(* CoDeSys 2.3 export: MODBUS_FBD.EXP *)

(* POU modbus_FBD, FBD *)
PROGRAM modbus_FBD
VAR
	get1_modbus: MB_RD_HOLD_REGS;    (*функция 03 - чтение параметра типа INT*)
	get2_modbus: MB_RD_INP_REGS;		(*функция 04 - чтение трех параметров типа INT*)
	get3_modbus: MB_RD_HOLD_REGS;	(*функция 03 - чтение параметра типа Float*)
	COM_SERVICE1: COM_SERVICE;		(*функция открытия COM-порта*)

	Buffer: ARRAY[0..255] OF BYTE;		(* байтовый буфер данных *)
     	cmpl: BOOL;
	port_opened:  BYTE := 0;
	Init: BOOL;								(* признак инициализации пользовательской программы *)
	Settings:COMSETTINGS;				(* настройки последовательного порта *)
      	com_num: PORTS:=0;				(*0 - RS-485, 1 - RS-232*)
	enabl: BOOL;							(*состояние работы блока*)
	err: INT;								(*номер ошибки*)
	TimeOut: TIME:=T#50ms;				(*таймаут*)
	Exception: BYTE;
	DataSize: WORD;
	master1: BYTE:= 0;

	x:WORD;						(*считанное значение*)
	x1: WORD;						(*переменная для записи по сети*)
	x2: WORD;						(*переменная для записи по сети*)
	x3: WORD;						(*переменная для записи по сети*)
	d:  REAL;						(*считанное значение*)
	ptr_D:POINTER TO BYTE;

	ctu1: CTU;
	a: BOOL;
	ynjj: BOOL;
END_VAR
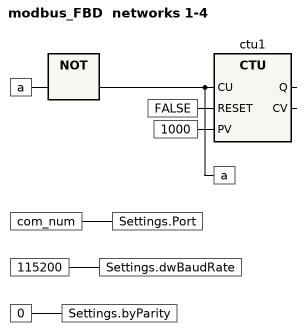
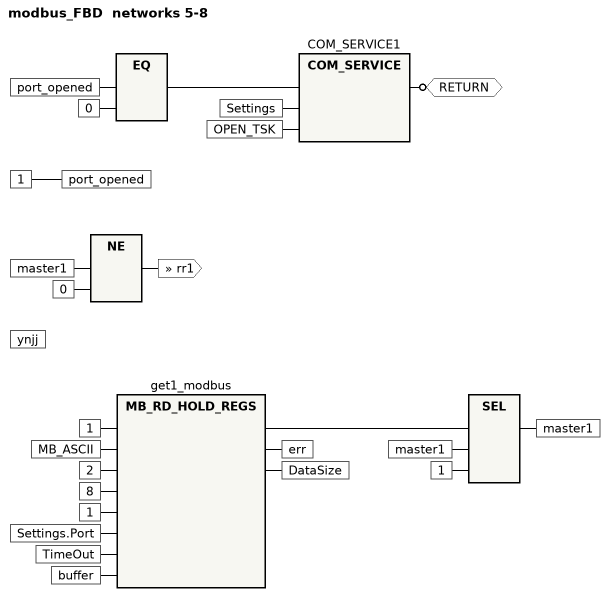
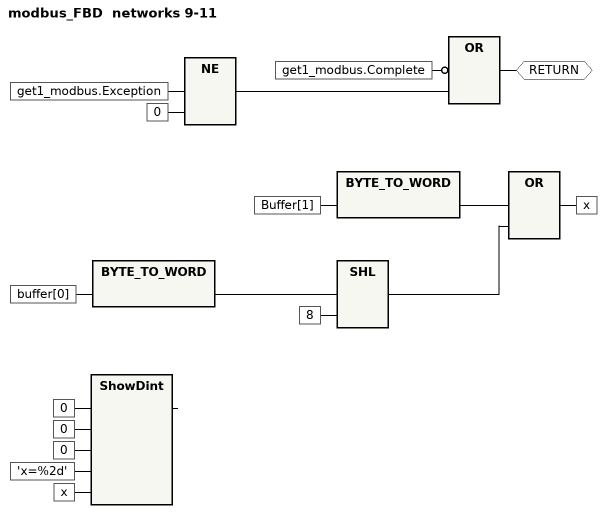
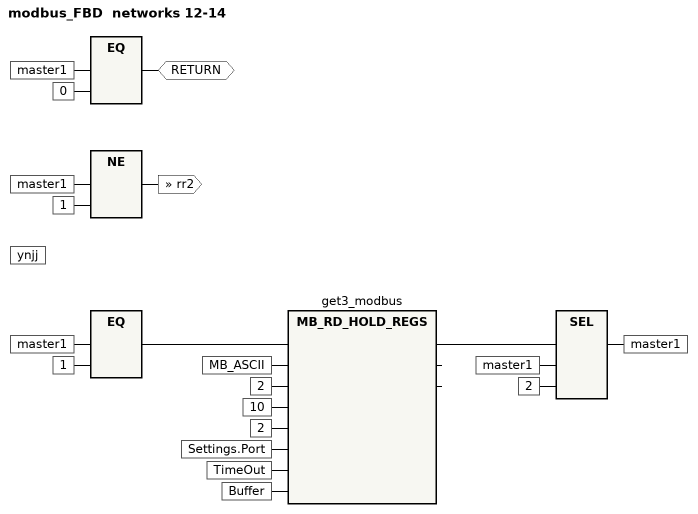
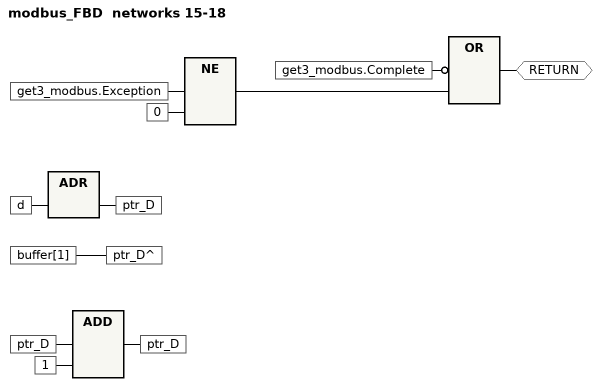
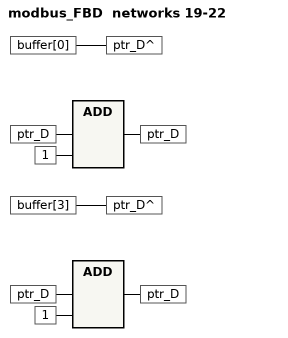
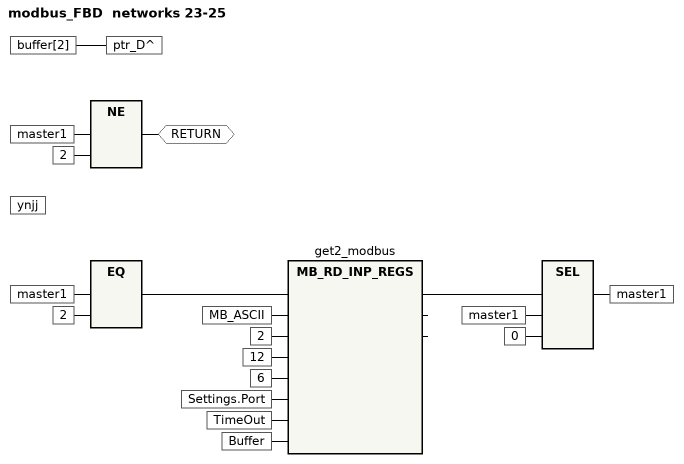
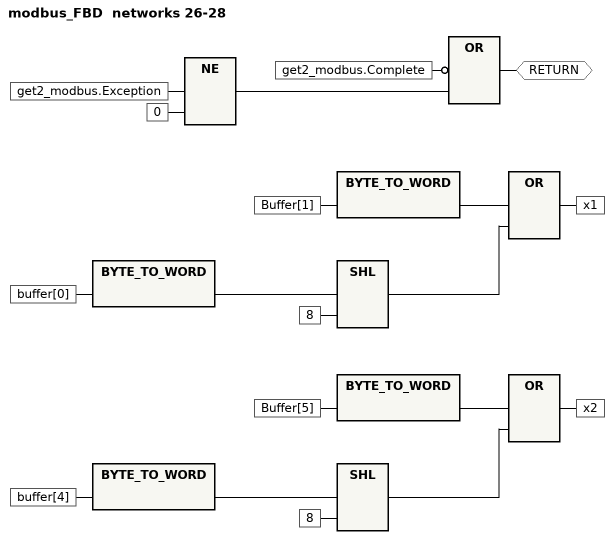
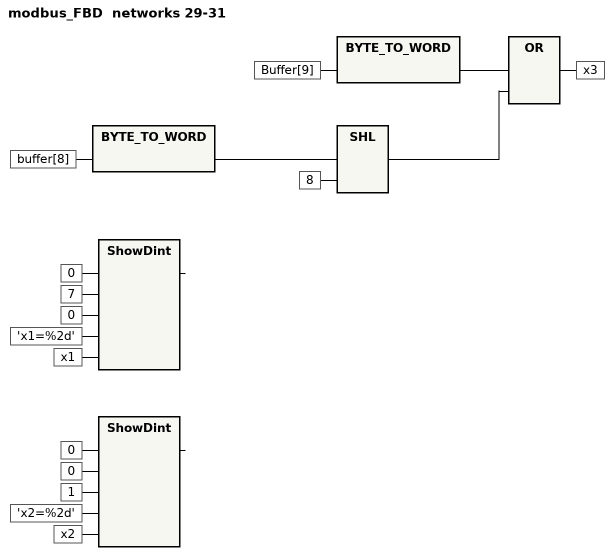
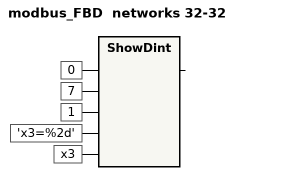
_FBD_ (* Function Block Diagram *)
NETWORK 1 (* Организуем счетчик, что бы передавать эти данные по сети *)
	ctu1:CTU(CU: <NOT(a) => a>, RESET: FALSE, PV: 1000)
NETWORK 2 (* ( *номер COM-порта* ) *)
	com_num => Settings.Port
NETWORK 3 (* ( *скорость* ) *)
	115200 => Settings.dwBaudRate
NETWORK 4 (* Кол-во стоповых бит 0 =один, 1=полтора , 2=два *)
	0 => Settings.byParity
NETWORK 5 (* ( *Открываем COM-порт* ) *)
	NOT COM_SERVICE1:COM_SERVICE(EQ(port_opened, 0), Settings, OPEN_TSK) => <RETURN>
NETWORK 6
	1 => port_opened
NETWORK 7
	NE(master1, 0) => >>rr1 => ynjj
NETWORK 8 (* ( * функция 03 инт  - ФБ считывает значение параметра  типа int из прибора с адресом 2 в регистр с номером 8 по протоколу Modbus-ASCII* ) *)
	SEL(get1_modbus:MB_RD_HOLD_REGS(1, MB_ASCII, 2, 8, 1, Settings.Port, TimeOut, buffer, out 2 => err, out 3 => DataSize), master1, 1) => master1
NETWORK 9
	OR(NOT get1_modbus.Complete, NE(get1_modbus.Exception, 0)) => <RETURN>
NETWORK 10
	OR(BYTE_TO_WORD(Buffer[1]), SHL(BYTE_TO_WORD(buffer[0]), 8)) => x
NETWORK 11
	ShowDint(0, 0, 0, 'x=%2d', x)
NETWORK 12
	EQ(master1, 0) => <RETURN>
NETWORK 13 rr1:
	NE(master1, 1) => >>rr2 => ynjj
NETWORK 14 (* ( * функция 03 флоат - ФБ считывает значение параметра  типа int из прибора с адресом 2 в регистр с номаром 10 по протоколу Modbus-ASCII * ) *)
	SEL(get3_modbus:MB_RD_HOLD_REGS(EQ(master1, 1), MB_ASCII, 2, 10, 2, Settings.Port, TimeOut, Buffer), master1, 2) => master1
NETWORK 15
	OR(NOT get3_modbus.Complete, NE(get3_modbus.Exception, 0)) => <RETURN>
NETWORK 16 (* получаем  данные из буфера типа FLOAT *)
	ADR(d) => ptr_D
NETWORK 17
	buffer[1] => ptr_D^
NETWORK 18
	ADD(ptr_D, 1) => ptr_D
NETWORK 19
	buffer[0] => ptr_D^
NETWORK 20
	ADD(ptr_D, 1) => ptr_D
NETWORK 21
	buffer[3] => ptr_D^
NETWORK 22
	ADD(ptr_D, 1) => ptr_D
NETWORK 23
	buffer[2] => ptr_D^
NETWORK 24 rr2:
	NE(master1, 2) => <RETURN> => ynjj
NETWORK 25 (* ( * функция 04 инт - ФБ считывает значения трех параметров типа Int из прибора с адресом 2 начиная с регистра с номeром 12* ) *)
	SEL(get2_modbus:MB_RD_INP_REGS(EQ(master1, 2), MB_ASCII, 2, 12, 6, Settings.Port, TimeOut, Buffer), master1, 0) => master1
NETWORK 26
	OR(NOT get2_modbus.Complete, NE(get2_modbus.Exception, 0)) => <RETURN>
NETWORK 27
	OR(BYTE_TO_WORD(Buffer[1]), SHL(BYTE_TO_WORD(buffer[0]), 8)) => x1
NETWORK 28
	OR(BYTE_TO_WORD(Buffer[5]), SHL(BYTE_TO_WORD(buffer[4]), 8)) => x2
NETWORK 29
	OR(BYTE_TO_WORD(Buffer[9]), SHL(BYTE_TO_WORD(buffer[8]), 8)) => x3
NETWORK 30
	ShowDint(0, 7, 0, 'x1=%2d', x1)
NETWORK 31
	ShowDint(0, 0, 1, 'x2=%2d', x2)
NETWORK 32
	ShowDint(0, 7, 1, 'x3=%2d', x3)
_END_FBD_
END_PROGRAM
